(* IEC 61131-3 sources: Industry-PLC-LLM/data/PLCBEAD_repo/PLCBEAD_PLCEmbed-main/PLC-BEAD/Source/GEB/building_SDD_NH3, 1 file *)

(* ---- SDD_NH3.ST ---- *)
FUNCTION SDD_NH3:REAL

	VAR_INPUT
		T :	REAL;
	END_VAR

	IF T < -33.65 THEN
		SDD_NH3 := EXP(7.3396511649 - ( 1166.7498002 / ( T + 192.37 )));
	ELSE
		SDD_NH3 := EXP(11.210964456 - ( 2564.9140075 / ( T + 262.741 )));
	END_IF;

END_FUNCTION

PROGRAM program0
  VAR
    T :	REAL;
    CEIL5_OUT : REAL;
  END_VAR

  CEIL5_OUT := SDD_NH3(T);
END_PROGRAM
